FUNCTION WristIK : REAL
VAR_INPUT
	
	// 末端坐标
	x: REAL;
	y: REAL;
	
END_VAR
VAR
	wrist_Axis_Angle	:REAL;	//腕关节角度
	
END_VAR


wrist_Axis_Angle := ACOS(y/(SQRT(x*x + y*y)));
IF x >= 0 THEN
	WristIK := RAD_TO_DEG(wrist_Axis_Angle);
ELSE
	WristIK := -RAD_TO_DEG(wrist_Axis_Angle);
END_IF

END_FUNCTION

(* stored: Version 1.1.0.1, ProductVersion 3.1.4024.14
   POU WristIK: Id {fa587cfb-998b-4872-b950-bf765eced708}, SpecialFunc None *)
